TYPE stSettings_Comm EXTENDS stSettings_Base :
STRUCT
	tConnectTimeout    : TIME := T#10S;
    tDisconnectTimeout : TIME := T#5S;
    tReconnectDelay    : TIME := T#2S;
    tStopTimeout       : TIME := T#10S;
    nMaxAutoReconnectAttempts : UINT := 3;
	
END_STRUCT
END_TYPE

(* stored: Version 1.1.0.1, ProductVersion 3.1.4026.18
   DUT stSettings_Comm: Id {399e18e4-e44f-4fbb-8c56-a1ad0a0061ec} *)
